// TIA Portal V15.1 export
// export: Created 2020-06-12T07:35:43.8662109Z, ExportSetting None, DisplayName Totally Integrated Automation Portal, DisplayVersion V15.1, DisplayName TIA Portal Openness, DisplayVersion V15.1, DisplayName STEP 7 Professional, DisplayVersion V15.1, DisplayName STEP 7 Safety, DisplayVersion V15.1, DisplayName WinCC Advanced, DisplayVersion V15.1
FUNCTION "PORT_call" : Void   // FC77, FBD
TITLE = Portal carriage call
{ S7_Optimized_Access := 'TRUE' }
// stored: SetENOAutomatically False
BEGIN

REGION Network 1: Movement
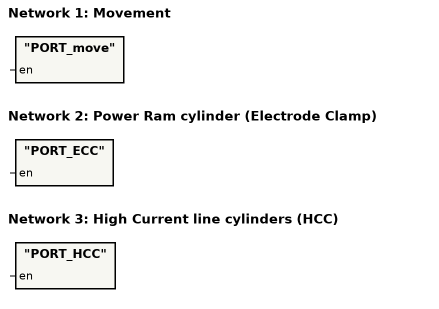
   "PORT_move"();
END_REGION

REGION Network 2: Power Ram cylinder (Electrode Clamp)
   "PORT_ECC"();
END_REGION

REGION Network 3: High Current line cylinders (HCC)
   "PORT_HCC"();
END_REGION
END_FUNCTION
